{attribute addProperty BoxType "AT2020-0250-0019"}
{attribute addProperty Id "ControlAT %Q*UINT1621Current_setpoint_value_ChAT %Q*ARRAY[0 ..14] OF INT240300"}
{attribute addProperty CRC "2624970934"}
{attribute addProperty SizeInBites "256"}
{attribute addProperty SizeInBytes "32"}
TYPE CC_Outputs_AA78E99F :
STRUCT
	{attribute addProperty Name "Control"}
	Control AT %Q* : UINT;
	{attribute addProperty Name "Current_setpoint_value_Ch"}
	Current_setpoint_value_Ch AT %Q* : ARRAY[0 ..14] OF INT;
END_STRUCT
END_TYPE

(* stored: Version 1.2.0.0, ProductVersion 3.1.4024.9
   DUT CC_Outputs_AA78E99F: Id {9c43e72b-78f6-410e-8ea5-e42cbea37bf9} *)
